TYPE "ModeOutStruct"
VERSION : 0.1
   STRUCT
      Estop : Bool;
      Reset : Bool;
      Manual : Bool;
      Auto : Bool;
      Home : Bool;
      Running : Bool;
      Change : Bool;
   END_STRUCT;

END_TYPE

